FUNCTION_BLOCK "G261M_Code"
TITLE =G261M BELT CONVEYOR 7200 KILN
//COPYRIGHT:    (C) 2009  BUHLER AG, CH-9240 UZWIL, SWITZERLAND
//
//PRODUCT:      WinCoS_BIW01_09
//
//TITLE:        BELT CONVEYOR 7200 KILN
//                Machine group control
//                Maschinengruppensteuerung
//
//--------------------------------------------------------------------------------
//
//IDENT:        AUTHOR:             DEPT:                              DATE:
//
//P01_FB361.1.0 K.Renz              CSB41                              08.Mrz.2010
//             1st Release
//
//--------------------------------------------------------------------------------
//
//PURPOSE:
//
//MANUAL :
//
//RESTRICTIONS:
//
//--------------------------------------------------------------------------------
AUTHOR : KR
FAMILY : USW
VERSION : 9.9


VAR
  Gr : "GCS7_GrpCtrlSub";	//Standard interface to group
  InOutValue1 : DINT ;	//Data for user
  InOutValue2 : DINT ;	//Data for user
  OutWayConflict : BOOL ;	//Data for user
  OutSelectionOk : BOOL ;	//Data for user
  CmdNewValue : BOOL ;	//Data for user
  CmdNewJob : BOOL ;	//Data for user
  OutCodeOK : BOOL ;	//Data for user
  InEndOfJob : BOOL ;	//Data for user
  staWayOk : BOOL ;	//Data for user
  EdgeStartRelease : BOOL ;	//Data for user
  USW8 : BOOL ;	//Data for user
  USW9 : BOOL ;	//Data for user
  USW10 : BOOL ;	//Data for user
  USW11 : BOOL ;	//Data for user
  USW12 : BOOL ;	//Data for user
  USW13 : BOOL ;	//Data for user
  USW14 : BOOL ;	//Data for user
  USW15 : BOOL ;	//Data for user
  A_2926_MXZ0MA : "A_2926_MXZ0MA_Code";	// Motor+6DI
  A_3101_KILN0 : "GCS7_E_DigInput";	// DigInpCont
  A_2926_QXV31 : "GCS7_E_ValveControl";	// VLS
END_VAR
VAR_TEMP
  tmpEnable : BOOL ;
  tmpFlag : BOOL ;
  tmpCmdNext : BOOL ;
  tmpLocal : BOOL ;
  tmpAspOk : BOOL ;
  tmpHWStop : BOOL ;
  tmpInstanzDBNo : INT ;
END_VAR
BEGIN
NETWORK
TITLE =



NETWORK
TITLE =Read command from group control
//Parameter
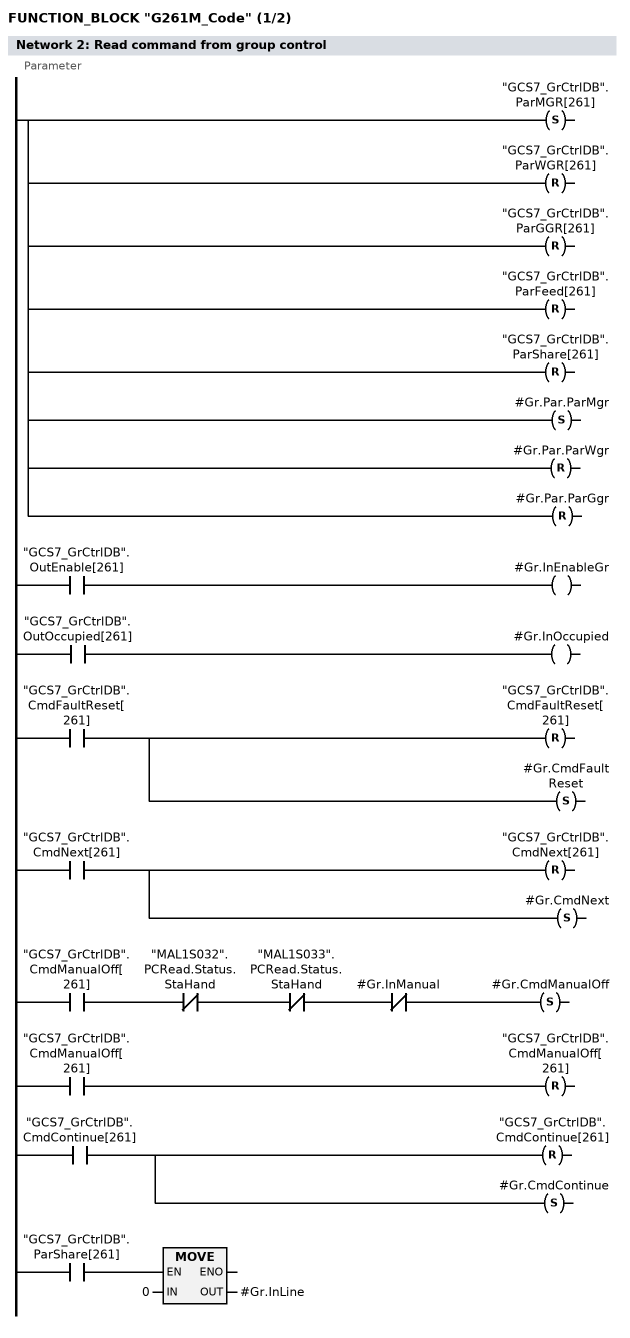
      SET   ;
      S     "GCS7_GrCtrlDB".ParMGR[261];
      R     "GCS7_GrCtrlDB".ParWGR[261];
      R     "GCS7_GrCtrlDB".ParGGR[261];
      R     "GCS7_GrCtrlDB".ParFeed[261];
      R     "GCS7_GrCtrlDB".ParShare[261];
      S     #Gr.Par.ParMgr;
      R     #Gr.Par.ParWgr;
      R     #Gr.Par.ParGgr;
//Command
      U     "GCS7_GrCtrlDB".OutEnable[261];
      =     #Gr.InEnableGr;
      U     "GCS7_GrCtrlDB".OutOccupied[261];
      =     #Gr.InOccupied;
      U     "GCS7_GrCtrlDB".CmdFaultReset[261];
      R     "GCS7_GrCtrlDB".CmdFaultReset[261];
      S     #Gr.CmdFaultReset;
      U     "GCS7_GrCtrlDB".CmdNext[261];
      R     "GCS7_GrCtrlDB".CmdNext[261];
      S     #Gr.CmdNext;

      U     "GCS7_GrCtrlDB".CmdManualOff[261];
      UN    "MAL1S032".PCRead.Status.StaHand;
      UN    "MAL1S033".PCRead.Status.StaHand;
      UN    #Gr.InManual;
      S     #Gr.CmdManualOff;
      U     "GCS7_GrCtrlDB".CmdManualOff[261];
      R     "GCS7_GrCtrlDB".CmdManualOff[261];

//      U     "GCS7_GrCtrlDB".CmdManualOff[261]
//      O     "GCS7_GrCtrlDB".OutOccupied[261]
//      R     "GCS7_GrCtrlDB".CmdManualOff[261]
//      S     #Gr.CmdManualOff

      U     "GCS7_GrCtrlDB".CmdContinue[261];
      R     "GCS7_GrCtrlDB".CmdContinue[261];
      S     #Gr.CmdContinue;
//Init Line Number
      U     "GCS7_GrCtrlDB".ParShare[261];
      SPBN  WE00;
      L     0;
      T     #Gr.InLine;
WE00: NOP   0;
NETWORK
TITLE =Call Methode Control
// 1. Handle Interface PCControl
// 2. Prepare mode --> ModePassive,ModeActive,ModeIdling
// 3. Reset global flags of the group
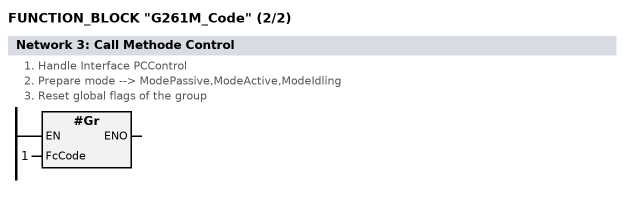
      CALL #Gr (
           FcCode                   := 1);
NETWORK
TITLE =Restart Idling Time

      L     #Gr.Par.ParIdling;
      L     2;
      >=I   ;
      SPB   IdTm;
      T     #Gr.Par.ParIdling;
IdTm: NOP   0;
      UN    "G284M".Gr.ModePassive;
      S     #Gr.CmdRestartIdling;
NETWORK
TITLE =Prepare global flags



NETWORK
TITLE =Set Pattern (Target position)



NETWORK
TITLE =Interlocking WayOk



NETWORK
TITLE =Interlocking Autostart
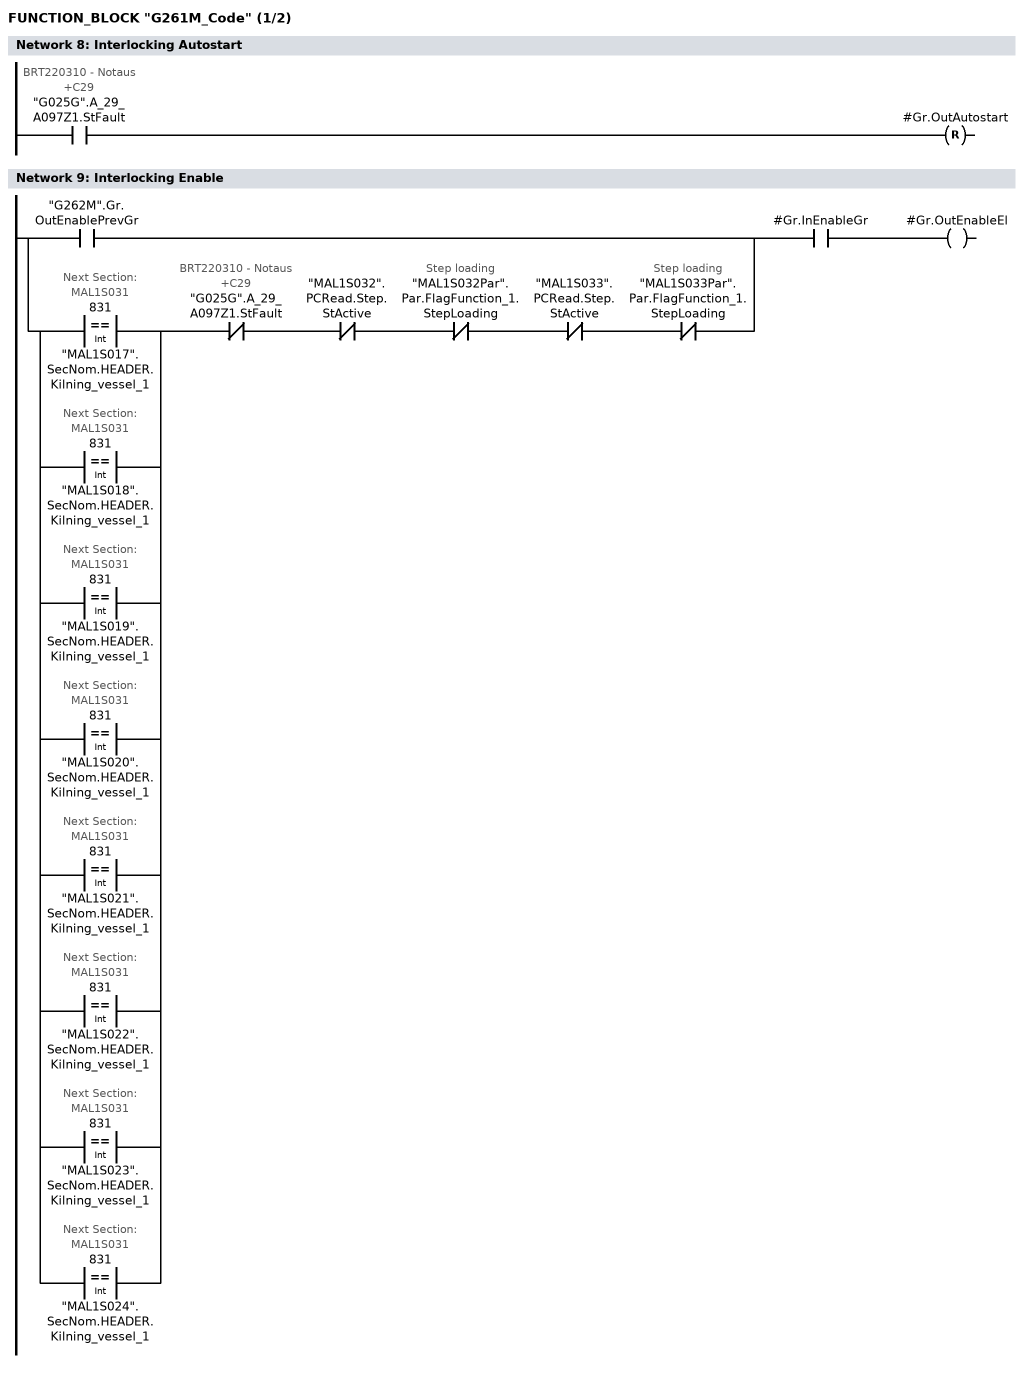

//      CLR
      U     "G025G".A_29_A097Z1.StFault; //BRT220310 - Notaus +C29
      R     #Gr.OutAutostart;
NETWORK
TITLE =Interlocking Enable

      U     "G262M".Gr.OutEnablePrevGr;
//KR10022010--->Wenn beladen Dummy Darre angewählt
      O(    ;
      O(    ;
      L     831; // Next Section: MAL1S031
      L     "MAL1S017".SecNom.HEADER.Kilning_vessel_1; // Target in recipe
      ==I   ;
      )     ;
//<---
//====>BRT190310
      O(    ;
      L     831; // Next Section: MAL1S031
      L     "MAL1S018".SecNom.HEADER.Kilning_vessel_1; // Target in recipe
      ==I   ;
      )     ;
      O(    ;
      L     831; // Next Section: MAL1S031
      L     "MAL1S019".SecNom.HEADER.Kilning_vessel_1; // Target in recipe
      ==I   ;
      )     ;
      O(    ;
      L     831; // Next Section: MAL1S031
      L     "MAL1S020".SecNom.HEADER.Kilning_vessel_1; // Target in recipe
      ==I   ;
      )     ;
      O(    ;
      L     831; // Next Section: MAL1S031
      L     "MAL1S021".SecNom.HEADER.Kilning_vessel_1; // Target in recipe
      ==I   ;
      )     ;
      O(    ;
      L     831; // Next Section: MAL1S031
      L     "MAL1S022".SecNom.HEADER.Kilning_vessel_1; // Target in recipe
      ==I   ;
      )     ;
      O(    ;
      L     831; // Next Section: MAL1S031
      L     "MAL1S023".SecNom.HEADER.Kilning_vessel_1; // Target in recipe
      ==I   ;
      )     ;
      O(    ;
      L     831; // Next Section: MAL1S031
      L     "MAL1S024".SecNom.HEADER.Kilning_vessel_1; // Target in recipe
      ==I   ;
      )     ;
      UN    "G025G".A_29_A097Z1.StFault; //BRT220310 - Notaus +C29
      UN    "MAL1S032".PCRead.Step.StActive;
      UN    "MAL1S032Par".Par.FlagFunction_1.StepLoading; // Step loading
      UN    "MAL1S033".PCRead.Step.StActive;
      UN    "MAL1S033Par".Par.FlagFunction_1.StepLoading; // Step loading
      )     ;
      U     #Gr.InEnableGr;
      =     #Gr.OutEnableEl;

NETWORK
TITLE =Interlocking Next
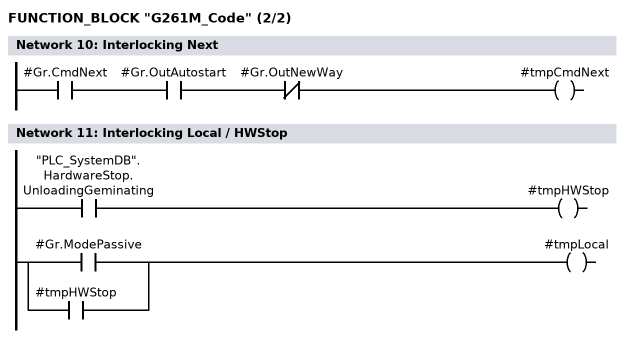

      U     #Gr.CmdNext;
      U     #Gr.OutAutostart;
      UN    #Gr.OutNewWay;
      =     #tmpCmdNext;

NETWORK
TITLE =Interlocking Local / HWStop

      U     "PLC_SystemDB".HardwareStop.UnloadingGeminating;
      =     #tmpHWStop;

      U     #Gr.ModePassive;
      O     #tmpHWStop;
      =     #tmpLocal;

NETWORK
TITLE =Interlocking Start Warning

      NOP   0;
//- Restart after fault --
      U     #Gr.CmdFaultReset;
      U     #Gr.VarFault;
      S     "SYS_StartWarningDB".Area[10].CmdResetStartWarning;
//- Run Timer --
      AUF   "G261M";
      CALL "GCS7_StartWarning" , "SYS_StartWarningDB" (
           InModeHigher             := FALSE,
           InArea                   := 10,
           InEnable                 := #Gr.OutEnableEl,
           InLocal                  := #tmpLocal,
           InStarted                := #Gr.VarStarted,
           InCmdNext                := #tmpCmdNext,
           OutCmdNext               := #tmpCmdNext,
           OutStartwarning          := #Gr.VarStartwarning);
//- Store Startwarning done  --
//- Reset Autostart --
      U     "SYS_StartWarningDB".TmpArea.OutStartReleaseRunningL;
      FN    #EdgeStartRelease;
      U     #Gr.VarFault;
      R     #Gr.OutAutostart;
NETWORK
TITLE ==A-2926-MXZ0MA : BELT CONVEYOR 7200
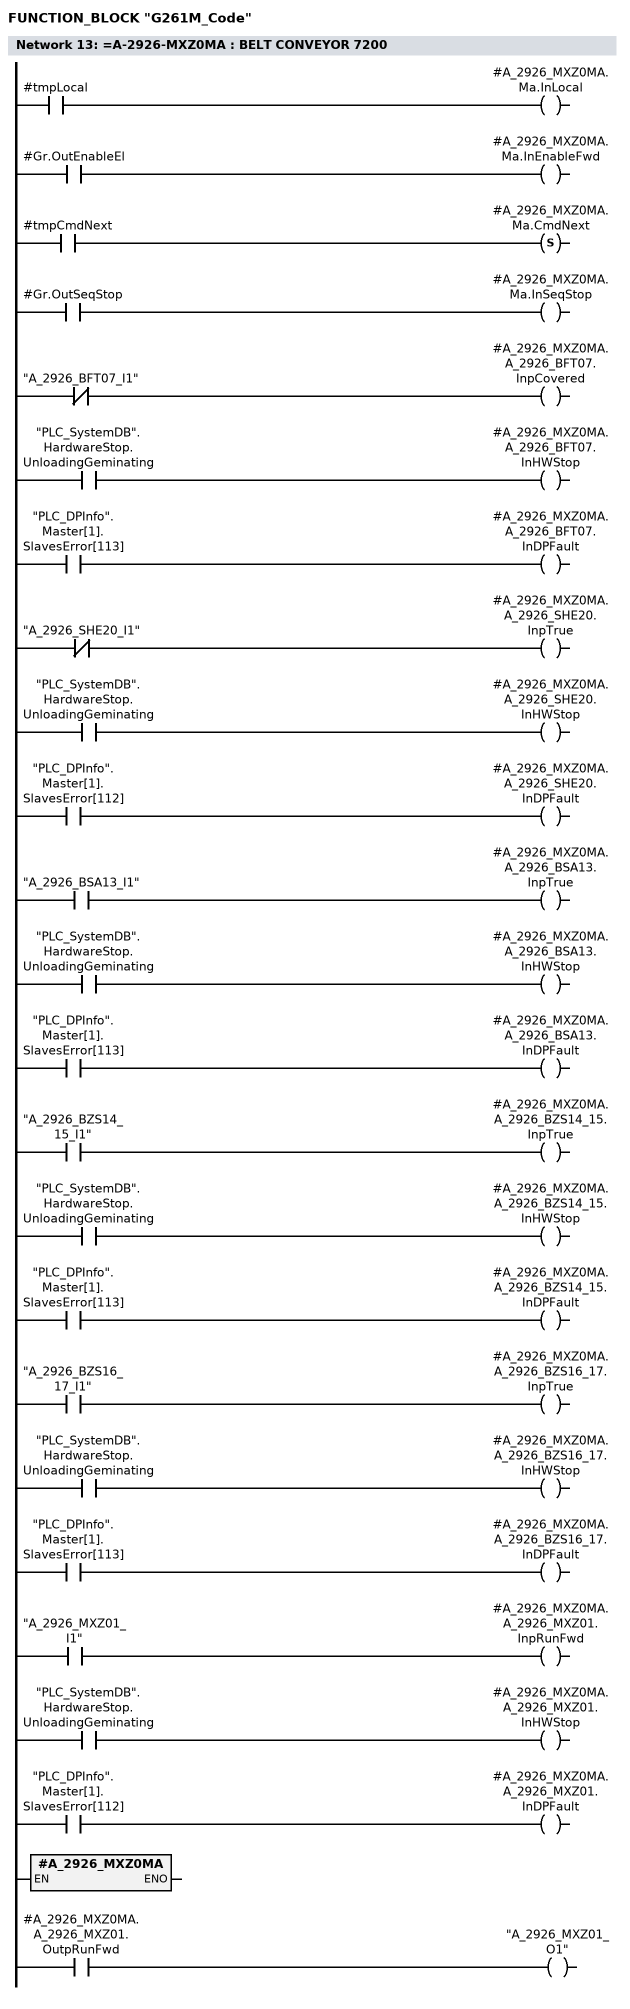

      NOP   0;
//-InLocal---
      U     #tmpLocal;
      =     #A_2926_MXZ0MA.Ma.InLocal;
//
//-Interlocking---

      U     #Gr.OutEnableEl;
      =     #A_2926_MXZ0MA.Ma.InEnableFwd;
//
      U     #tmpCmdNext;
      S     #A_2926_MXZ0MA.Ma.CmdNext;
//
      U     #Gr.OutSeqStop;
      =     #A_2926_MXZ0MA.Ma.InSeqStop;
//
//=Values and commands of elements===
//-=A-2926-BFT07---
//      CLR
//      S     #A_2926_MXZ0MA.A_2926_BFT07.CmdRunTimeOutTime
//-=A-2926-SHE20---
//      CLR
//      S     #A_2926_MXZ0MA.A_2926_SHE20.CmdRunTimeOutTime
//-=A-2926-BSA13---
//      CLR
//      S     #A_2926_MXZ0MA.A_2926_BSA13.CmdRunTimeOutTime
//-=A-2926-BZS14/15---
//      CLR
//      S     #A_2926_MXZ0MA.A_2926_BZS14_15.CmdRunTimeOutTime
//-=A-2926-BZS16/17---
//      CLR
//      S     #A_2926_MXZ0MA.A_2926_BZS16_17.CmdRunTimeOutTime
//
//-Read inputs of elements---
      UN    "A_2926_BFT07_I1";
      =     #A_2926_MXZ0MA.A_2926_BFT07.InpCovered;
      U     "PLC_SystemDB".HardwareStop.UnloadingGeminating;
      =     #A_2926_MXZ0MA.A_2926_BFT07.InHWStop;
      U     "PLC_DPInfo".Master[1].SlavesError[113];
      =     #A_2926_MXZ0MA.A_2926_BFT07.InDPFault;
//BRT080310      U     "A_2926_SHE20_I1"
      UN    "A_2926_SHE20_I1";
      =     #A_2926_MXZ0MA.A_2926_SHE20.InpTrue;
      U     "PLC_SystemDB".HardwareStop.UnloadingGeminating;
      =     #A_2926_MXZ0MA.A_2926_SHE20.InHWStop;
      U     "PLC_DPInfo".Master[1].SlavesError[112];
      =     #A_2926_MXZ0MA.A_2926_SHE20.InDPFault;
      U     "A_2926_BSA13_I1";
      =     #A_2926_MXZ0MA.A_2926_BSA13.InpTrue;
      U     "PLC_SystemDB".HardwareStop.UnloadingGeminating;
      =     #A_2926_MXZ0MA.A_2926_BSA13.InHWStop;
      U     "PLC_DPInfo".Master[1].SlavesError[113];
      =     #A_2926_MXZ0MA.A_2926_BSA13.InDPFault;
      U     "A_2926_BZS14_15_I1";
      =     #A_2926_MXZ0MA.A_2926_BZS14_15.InpTrue;
      U     "PLC_SystemDB".HardwareStop.UnloadingGeminating;
      =     #A_2926_MXZ0MA.A_2926_BZS14_15.InHWStop;
      U     "PLC_DPInfo".Master[1].SlavesError[113];
      =     #A_2926_MXZ0MA.A_2926_BZS14_15.InDPFault;
      U     "A_2926_BZS16_17_I1";
      =     #A_2926_MXZ0MA.A_2926_BZS16_17.InpTrue;
      U     "PLC_SystemDB".HardwareStop.UnloadingGeminating;
      =     #A_2926_MXZ0MA.A_2926_BZS16_17.InHWStop;
      U     "PLC_DPInfo".Master[1].SlavesError[113];
      =     #A_2926_MXZ0MA.A_2926_BZS16_17.InDPFault;
      U     "A_2926_MXZ01_I1";
      =     #A_2926_MXZ0MA.A_2926_MXZ01.InpRunFwd;
      U     "PLC_SystemDB".HardwareStop.UnloadingGeminating;
      =     #A_2926_MXZ0MA.A_2926_MXZ01.InHWStop;
      U     "PLC_DPInfo".Master[1].SlavesError[112];
      =     #A_2926_MXZ0MA.A_2926_MXZ01.InDPFault;
//
//-Set Parameters---
//
//-Call object control---
      CALL #A_2926_MXZ0MA ;
//
//-Write outputs---
      U     #A_2926_MXZ0MA.A_2926_MXZ01.OutpRunFwd;
      =     "A_2926_MXZ01_O1";
NETWORK
TITLE ==A-3101-KILN0 : SIGNAL ALTE DARRE INFEEDING

      NOP   0;
//-InLocal---
      U     #tmpLocal;
      =     #A_3101_KILN0.InLocal;
//
//-Monitoring---
      CLR   ;
      =     #A_3101_KILN0.InMonTrue;
      CLR   ;
      =     #A_3101_KILN0.InMonFalse;
//
//-PreAlarm---
      CLR   ;
      =     #A_3101_KILN0.InPreAlarmTrue;
      CLR   ;
      =     #A_3101_KILN0.InPreAlarmFalse;
//
//-Additional commands---
//      CLR
//      S     #A_3101_KILN0.CmdRunTimeOutTime
//
//-Read inputs---
      U     "A_3101_KILN0_I1";
      =     #A_3101_KILN0.InpTrue;
      U     "PLC_DPInfo".Master[1].SlavesError[112];
      =     #A_3101_KILN0.InDPFault;
//
//-Set Parameters---
//
//-Call object control---
      CALL #A_3101_KILN0 ;
//
//-Write outputs---
NETWORK
TITLE ==A-2926-QXV31 : BALL VALVE SPRAY WATER OPEN

      NOP   0;
//-InLocal---
      U     #tmpLocal;
      =     #A_2926_QXV31.InLocal;
//
//-Interlocking---
      U     #A_2926_MXZ0MA.Ma.StStartedFwd;
      =     #A_2926_QXV31.InEnableHN;
      NOT   ;
      =     #A_2926_QXV31.InEnableLN;
//
      SET   ;
      S     #A_2926_QXV31.CmdNext;
//
      U     #Gr.OutSeqStop;
      =     #A_2926_QXV31.InSeqStop;
//
//-Read inputs---
      UN    #A_2926_QXV31.OutpHN;
      =     #A_2926_QXV31.InpLN;
      U     #A_2926_QXV31.OutpHN;
      =     #A_2926_QXV31.InpHN;
      U     "PLC_SystemDB".HardwareStop.UnloadingGeminating;
      =     #A_2926_QXV31.InHWStop;
      U     "PLC_DPInfo".Master[1].SlavesError[113];
      =     #A_2926_QXV31.InDPFault;
//
//-Set Parameters---
//
//-Call object control---
      CALL #A_2926_QXV31 ;
//
//-Write outputs---
      U     #A_2926_QXV31.OutpHN;
      =     "A_2926_QXV31_O1";
NETWORK
TITLE =Test Fault

      U     #A_2926_MXZ0MA.Ma.StFault;
      O     #A_3101_KILN0.StFault;
      O     #A_2926_QXV31.StFault;
      =     #Gr.VarFault;
NETWORK
TITLE =Test Warning

      CLR   ;
      =     #Gr.OutWarning;
NETWORK
TITLE =Test Stopped
//BRT080310      U     #A_2926_MXZ0MA.Ma.StStopped
//BRT080310      UN    #Gr.VarFault
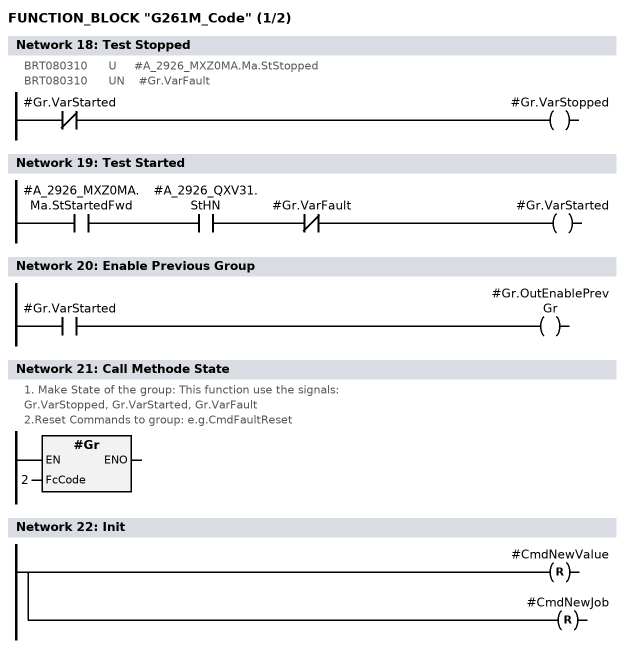
      UN    #Gr.VarStarted;
      =     #Gr.VarStopped;
NETWORK
TITLE =Test Started

      U     #A_2926_MXZ0MA.Ma.StStartedFwd;
//BRT080310      UN    #Gr.VarStopped
      U     #A_2926_QXV31.StHN;
      UN    #Gr.VarFault;
      =     #Gr.VarStarted;
NETWORK
TITLE =Enable Previous Group

      U     #Gr.VarStarted;
      =     #Gr.OutEnablePrevGr;
NETWORK
TITLE =Call Methode State
//1. Make State of the group: This function use the signals:
//        Gr.VarStopped, Gr.VarStarted, Gr.VarFault
//2.Reset Commands to group: e.g.CmdFaultReset
      CALL #Gr (
           FcCode                   := 2);
NETWORK
TITLE =Init

      SET   ;
      R     #CmdNewValue;
      R     #CmdNewJob;
NETWORK
TITLE =Write data to group control
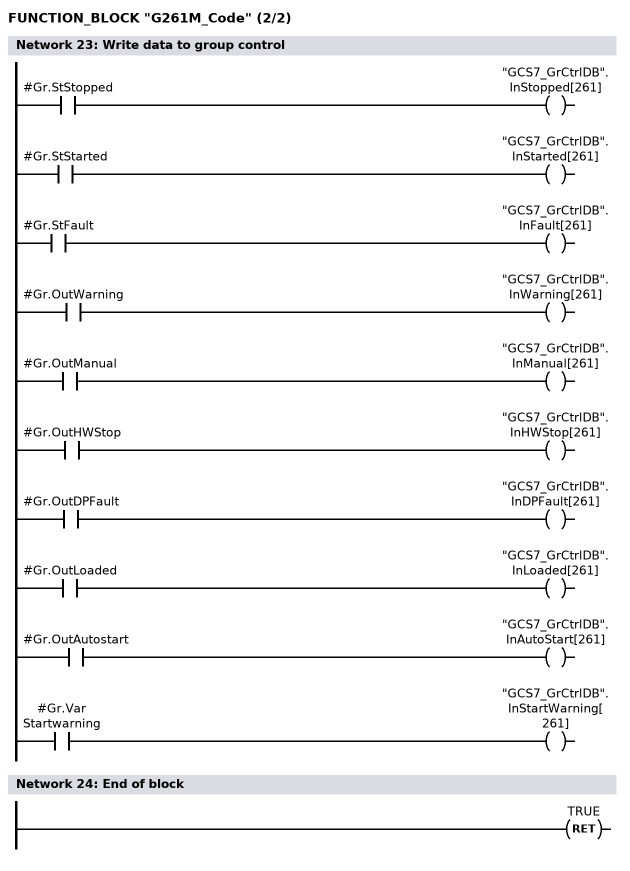

      U     #Gr.StStopped;
      =     "GCS7_GrCtrlDB".InStopped[261];
      U     #Gr.StStarted;
      =     "GCS7_GrCtrlDB".InStarted[261];
      U     #Gr.StFault;
      =     "GCS7_GrCtrlDB".InFault[261];
      U     #Gr.OutWarning;
      =     "GCS7_GrCtrlDB".InWarning[261];
      U     #Gr.OutManual;
      =     "GCS7_GrCtrlDB".InManual[261];
      U     #Gr.OutHWStop;
      =     "GCS7_GrCtrlDB".InHWStop[261];
      U     #Gr.OutDPFault;
      =     "GCS7_GrCtrlDB".InDPFault[261];
      U     #Gr.OutLoaded;
      =     "GCS7_GrCtrlDB".InLoaded[261];
      U     #Gr.OutAutostart;
      =     "GCS7_GrCtrlDB".InAutoStart[261];
      U     #Gr.VarStartwarning;
      =     "GCS7_GrCtrlDB".InStartWarning[261];
NETWORK
TITLE =End of block

      BE    ;

END_FUNCTION_BLOCK

